{region '#Template'}
	{attribute 'Version' := '1.0.0.0'}
	{attribute 'Tags' := '"LCID": "1031", "Text": "DUT, System, UPS"'}
	{attribute 'Tags' := '"LCID": "1033", "Text": "DUT, System, UPS"'}
	{attribute 'Description' := '"LCID": "1031", "Text": "Einstellung USV"'}
	{attribute 'Description' := '"LCID": "1033", "Text": "Settings UPS"'}
{endregion}

{attribute 'qualified_only'}
{attribute 'strict'}
TYPE E_BA_UPSType :
(
	eNone := 0,
	
	eCX50x0,
	eCX51x0,
	eCX81xx,
	eCX9020_U900,
	eCB3011
);
END_TYPE

(* stored: Version 1.1.0.1, ProductVersion 3.1.4024.9
   DUT E_BA_UPSType: Id {85020888-b87a-4539-84d0-da87fa089f9a} *)
